// TwinCAT 3 PLC project TcpIp_SERVER_with_TLS_PSK
// Title: TLS Sample
// Company: Beckhoff Automation
// ProjectVersion: 1.0.0.0
// ProgramVersion: 3.1.0.5
// libraries:
//   Tc2_Standard, * (Beckhoff Automation GmbH)
//   Tc2_System, * (Beckhoff Automation GmbH)
//   Tc2_TcpIp, * (Beckhoff Automation GmbH)
//   Tc2_Utilities, * (Beckhoff Automation GmbH)
//   Tc3_Module, * (Beckhoff Automation GmbH)
// project tree:
//   Data types/ E_ConnectionSteps.TcDUT (not stored), E_ServerSteps.TcDUT
//   Global Variables/ Global_Variables.TcGVL
//   POUs/ FB_Server.TcPOU, FB_ServerApplication.TcPOU, FB_ServerConnection.TcPOU, MAIN.TcPOU
//   POUs/Helper POUs/ FB_FrameFifo.TcPOU (not stored), FB_LogFifo.TcPOU (not stored), FB_TlsConfig.TcPOU
//   / PlcTaskServer.TcTTO
// real-time tasks:
//   TASK PlcTaskServer: cycle T#10ms, priority 20, ADS port 350

CONFIGURATION TcpIp_SERVER_with_TLS_PSK
    RESOURCE PLC ON TwinCAT3
        TASK PlcTaskServer(INTERVAL := T#10ms, PRIORITY := 20);
        PROGRAM MAIN WITH PlcTaskServer : MAIN;
    END_RESOURCE
END_CONFIGURATION

// ---- Data types/E_ServerSteps.TcDUT
TYPE E_ServerSteps :
(
	eSERVER_STATE_IDLE,
	eSERVER_STATE_SOCKET_CREATE,
	eSERVER_STATE_LISTENER_OPEN_START,
	eSERVER_STATE_LISTENER_OPEN_WAIT,
	eSERVER_STATE_REMOTE_CLIENTS_COMM,
	eSERVER_STATE_REMOTE_CLIENTS_CLOSE,
	eSERVER_STATE_LISTENER_CLOSE_START,
	eSERVER_STATE_LISTENER_CLOSE_WAIT,
	eSERVER_STATE_ERROR
);
END_TYPE

// ---- Global Variables/Global_Variables.TcGVL
VAR_GLOBAL CONSTANT
	MAX_CLIENT_CONNECTIONS					: UDINT(1..20) := 5;
	PLCPRJ_BUFFER_SIZE						: UDINT := 1000;(* Max. internal fifo/receiver buffer size *)

(*	PLCPRJ_CLIENT_SEND_CYCLE_TIME			: TIME := T#1S; not used at server side *)
	PLCPRJ_RECEIVE_POLLING_TIME				: TIME := T#100MS;
	PLCPRJ_RECEIVE_TIMEOUT					: TIME := T#50S;

	(* Some project specific error codes *)
	PLCPRJ_ERROR_RECEIVE_TIMEOUT			: UDINT := 16#8101;(* Receive timeout *)
	PLCPRJ_ERROR_SENDFIFO_OVERFLOW			: UDINT := 16#8102;(* Send fifo overflow *)
	PLCPRJ_ERROR_RECFIFO_OVERFLOW			: UDINT := 16#8103;(* Receive fifo overflow *)
END_VAR

// ---- POUs/MAIN.TcPOU
PROGRAM MAIN
VAR
	sSrvNetID   : T_AmsNetID :='';(* TwinCAT TCP/IP server network address *)
	{warning 'Please configure your server IP-address and server port number below:'}
	sLocalHost  : T_IPv4Addr :='127.0.0.1';(*Own (server) IP address! *)
	nLocalPort  : UINT       :=200;(* Own (server) port number! *)
	
	bEnable     : BOOL       :=TRUE;(* TRUE => Enable server data exchange, FALSE => Disable *)
	bLog        : BOOL       :=TRUE;(* TRUE => Enable message/error log, FALSE => Disable *)
	
	bPSK        : BOOL       :=TRUE;(* TRUE => use PSK , FALSE => don't use PSK *)
	key         : ARRAY[0..14] OF BYTE:=[16#1B,16#D0,16#6F,16#D2,16#56,16#16,16#7D,16#C1,16#E8,16#C7,16#48,16#2A,16#8E,16#F5,16#FF];
	fbTls       : FB_TlsConfig;(* TLS/PSK configuration *)
	
	fbServer    : FB_Server:=(sLocalHost:=sLocalHost, nLocalPort:=nLocalPort, sPrefix:='SERVER::');
	fbCloseAll  : FB_SocketCloseAll;
	bInitialize : BOOL:=TRUE;
END_VAR

IF bInitialize THEN
	(* On PLC reset or program download close all created/opened sockets/connections *)
	fbCloseAll(sSrvNetID:=sSrvNetID, bExecute:=bInitialize);
	IF fbCloseAll.bBusy OR fbCloseAll.bError THEN
		RETURN;
	END_IF
	
	(* Configure TLS/PSK settings *)
	fbTls.Clear();
	IF bPSK THEN
		fbTls.AddPsk(key:=key, sIdentity:='MyIdentity');
	END_IF
	
	bInitialize:=FALSE;
END_IF

fbServer(fbTls:=fbTls, sSrvNetID:=sSrvNetID, bEnable:=bEnable, bLog:=bLog);

END_PROGRAM

// ---- POUs/Helper POUs/FB_TlsConfig.TcPOU
(* TLS/PSK configuration *)
{attribute 'no_explicit_call':='Direct call not allowed for type FB_TlsConfig'}
{attribute 'no_assign'}
FUNCTION_BLOCK FB_TlsConfig
VAR
	_pskKey       : ARRAY[0..TCPADS_TLS_MAX_PSK_KEY_SIZE] OF BYTE;
	_pskKeyLen    : UDINT:=0;
	_sIdentity    : STRING(TCPADS_TLS_PSK_IDENTITY_SIZE);
	_sCaPath      : STRING(TCPADS_TLS_CERTIFICATE_PATH_SIZE);
	_sCrlPath     : STRING(TCPADS_TLS_CERTIFICATE_PATH_SIZE);
	_sCertPath    : STRING(TCPADS_TLS_CERTIFICATE_PATH_SIZE);
	_sKeyPath     : STRING(TCPADS_TLS_CERTIFICATE_PATH_SIZE);
	_sKeyPwd      : STRING(TCPADS_TLS_KEY_PASSWORD_SIZE);
	_listenFlags  : ST_TlsListenFlags:=DEFAULT_TLSLISTENFLAGS;
	_connectFlags : ST_TlsConnectFlags:=DEFAULT_TLSCONNECTFLAGS;
END_VAR

(* Adds CA certificate path *)
METHOD FINAL AddCa
VAR_INPUT
	sCaPath : STRING(TCPADS_TLS_CERTIFICATE_PATH_SIZE);
END_VAR
_sCaPath:=sCaPath;
END_METHOD

(* Adds certificate path *)
METHOD FINAL AddCert
VAR_INPUT
	sCertPath: STRING(TCPADS_TLS_CERTIFICATE_PATH_SIZE);
	sKeyPath: STRING(TCPADS_TLS_CERTIFICATE_PATH_SIZE);
	sKeyPwd: STRING(TCPADS_TLS_KEY_PASSWORD_SIZE);
END_VAR
_sCertPath:=sCertPath;
_sKeyPath:=sKeyPath;
_sKeyPwd:=sKeyPwd;
END_METHOD

METHOD FINAL AddConnectFlags
VAR_INPUT
	flags : ST_TlsConnectFlags;
END_VAR
_connectFlags:=flags;
END_METHOD

(* Adds certificate revocation list path *)
METHOD FINAL AddCrl
VAR_INPUT
	sCrlPath : STRING(TCPADS_TLS_CERTIFICATE_PATH_SIZE);
END_VAR
_sCrlPath:=sCrlPath;
END_METHOD

METHOD FINAL AddListenFlags
VAR_INPUT
	flags : ST_TlsListenFlags;
END_VAR
_listenFlags:=flags;
END_METHOD

(* Adds PSK and PSK identity *)
METHOD FINAL AddPsk
VAR_IN_OUT
	key : ARRAY[*] OF BYTE;
END_VAR
VAR_INPUT
	sIdentity : STRING(TCPADS_TLS_PSK_IDENTITY_SIZE);
END_VAR
_pskKeyLen:=MIN(DINT_TO_UDINT(UPPER_BOUND(key, 1) - LOWER_BOUND(key, 1) + 1), TCPADS_TLS_MAX_PSK_KEY_SIZE, SIZEOF(_pskKey));
MEMCPY(ADR(_pskKey[0]), ADR(key[LOWER_BOUND(key, 1)]), _pskKeyLen);
_sIdentity:=sIdentity;
END_METHOD

METHOD FINAL Clear
_sIdentity:='';
_pskKeyLen:=0;
MEMSET(ADR(_pskKey[0]), 0, SIZEOF(_pskKey));
_sCaPath:='';
_sCertPath:='';
_sKeyPath:='';
_sKeyPwd:='';
_sCrlPath:='';
END_METHOD

PROPERTY FINAL connectFlags : ST_TlsConnectFlags
GET
connectFlags:=_connectFlags;
END_GET
END_PROPERTY

PROPERTY FINAL listenFlags : ST_TlsListenFlags
GET
listenFlags:=_listenFlags;
END_GET
END_PROPERTY

(* Pointer to first PSK key byte *)
PROPERTY FINAL pskKey : PVOID
GET
pskKey:=SEL(_pskKeyLen = 0, ADR(_pskKey[0]), 0);
END_GET
END_PROPERTY

(* Byte size of PSK key *)
PROPERTY FINAL pskKeyLen : UDINT(0..TCPADS_TLS_MAX_PSK_KEY_SIZE)
GET
pskKeyLen:=_pskKeyLen;
END_GET
END_PROPERTY

(* CA certificate path *)
PROPERTY FINAL sCaPath : STRING(TCPADS_TLS_CERTIFICATE_PATH_SIZE)
GET
sCaPath:=_sCaPath;
END_GET
END_PROPERTY

(* Certificate path *)
PROPERTY FINAL sCertPath : STRING(TCPADS_TLS_CERTIFICATE_PATH_SIZE)
GET
sCertPath:=_sCertPath;
END_GET
END_PROPERTY

(* Certificate revocation list path *)
PROPERTY FINAL sCrlPath : STRING(TCPADS_TLS_CERTIFICATE_PATH_SIZE)
GET
sCrlPath:=_sCrlPath;
END_GET
END_PROPERTY

(* PSK key identity *)
PROPERTY FINAL sIdentity : STRING(TCPADS_TLS_PSK_IDENTITY_SIZE)
GET
sIdentity:=_sIdentity;
END_GET
END_PROPERTY

(* Certificate key path *)
PROPERTY FINAL sKeyPath : STRING(TCPADS_TLS_CERTIFICATE_PATH_SIZE)
GET
sKeyPath:=_sKeyPath;
END_GET
END_PROPERTY

(* Certificate key password *)
PROPERTY FINAL sKeyPwd : STRING(TCPADS_TLS_KEY_PASSWORD_SIZE)
GET
sKeyPwd:=_sKeyPwd;
END_GET
END_PROPERTY

END_FUNCTION_BLOCK

// ---- POUs/FB_Server.TcPOU
FUNCTION_BLOCK FB_Server
VAR_IN_OUT
	fbTls          : FB_TlsConfig;(* TLS/PSK configuration *)
END_VAR
VAR_INPUT
	sSrvNetID      : T_AmsNetID :='';(* TwinCAT TCP/IP server network address *)
	sLocalHost     : T_IPv4Addr :='127.0.0.1';(* Own IP address! *)
	nLocalPort     : UDINT      :=0;(* Server port number *)
	bEnable        : BOOL       :=FALSE;(* TRUE => enable server data exchange, FALSE => disable *)
	tReconnect     : TIME       :=T#3S;(* Reopen new listener socket after this time *)
	bLog           : BOOL       :=FALSE;(* TRUE => Enable log message output, FALSE => Disable *)
	sPrefix        : STRING     :='SERVER::';(* Log message description string (allows the identification of log message source) *)
END_VAR
VAR_OUTPUT
	bListening     : BOOL       :=FALSE;(* Listener socket state *)
	nAccepted      : UDINT      :=0;(* Max. number of accepted client connections *)
END_VAR
VAR
	aApplications  : ARRAY[1..MAX_CLIENT_CONNECTIONS] OF FB_ServerApplication;(* Server application control function blocks *)
	aConnections   : ARRAY[1..MAX_CLIENT_CONNECTIONS] OF FB_ServerConnection :=[
														(sPrefix := 'SERVER1::'),
														(sPrefix := 'SERVER2::'),
														(sPrefix := 'SERVER3::'),
														(sPrefix := 'SERVER4::'),
														(sPrefix := 'SERVER5::')];(* Server connection/data exchange control function blocks *)
	aTx            : ARRAY[1..MAX_CLIENT_CONNECTIONS] OF FB_FrameFifo;(* TX fifo *)
	aRx            : ARRAY[1..MAX_CLIENT_CONNECTIONS] OF FB_FrameFifo;(* RX fifo *)
	aLog           : ARRAY[1..MAX_CLIENT_CONNECTIONS] OF FB_LogFifo;(* Listener log message fifo *)

	fbCreate       : FB_TlsSocketCreate:=(bListener:=TRUE);(* Creates listener socket *)
	fbListen       : FB_TlsSocketListen;(* Opens listener socket *)
	fbSetPsk       : FB_TlsSocketSetPsk;(* Configures PSK (pre-shared key) *)
	fbClose        : FB_SocketClose;(* Closes socket *)
	fbLog          : FB_LogFifo;
	fbListenTimer  : TON;
	bReset         : BOOL :=FALSE;
	eStep          : E_ServerSteps;
	i              : UDINT;
END_VAR

CASE eStep OF
	eSERVER_STATE_IDLE:
		IF bEnable XOR bListening THEN
			IF bEnable THEN
				fbListenTimer( IN := TRUE );
				IF fbListenTimer.Q THEN
					fbListenTimer( IN := FALSE, PT := tReconnect );

					fbLog.Clear( sPrefix := sPrefix, bLog := bLog );(* Clear listener log fifo *)
					bReset := FALSE;

					fbCreate(bExecute:=FALSE);
					fbCreate(sSrvNetID:=sSrvNetID, bExecute:=TRUE);
					eStep := eSERVER_STATE_SOCKET_CREATE;
				END_IF
			ELSE
				eStep := eSERVER_STATE_REMOTE_CLIENTS_CLOSE;
			END_IF
		ELSIF bListening THEN
			eStep := eSERVER_STATE_REMOTE_CLIENTS_COMM;
		ELSE
			fbListenTimer( IN := FALSE, PT := T#0S );
			bReset := FALSE;
		END_IF
		
	eSERVER_STATE_SOCKET_CREATE:
		fbCreate(bExecute:=FALSE);
		IF NOT fbCreate.bBusy THEN
			IF NOT fbCreate.bError THEN
				fbSetPsk(bExecute:=FALSE);
				IF (fbTls.pskKeyLen <> 0) AND (fbTls.pskKey <> 0) AND (fbTls.sIdentity <> '') THEN
					fbSetPsk(sSrvNetID:=sSrvNetID, hSocket:=fbCreate.hSocket, sIdentity:=fbTls.sIdentity, pskKey:=fbTls.pskKey, pskKeyLen:=fbTls.pskKeyLen, bExecute:=TRUE);
				END_IF
				eStep := eSERVER_STATE_LISTENER_OPEN_START;
			ELSE
				fbLog.Error( sMessage := 'FB_TlsSocketCreate()', nErrId := fbCreate.nErrId);
				eStep := eSERVER_STATE_ERROR;
			END_IF
		END_IF

	eSERVER_STATE_LISTENER_OPEN_START:
		fbSetPsk(bExecute:=FALSE);
		IF NOT fbSetPsk.bBusy THEN
			IF NOT fbSetPsk.bError THEN
				fbListen(bExecute:=FALSE, hListener:=fbCreate.hSocket);
				fbListen(sSrvNetID:=sSrvNetID, bExecute:=TRUE, hListener:=fbCreate.hSocket, sLocalHost:=sLocalHost, nLocalPort:=nLocalPort);
				eStep := eSERVER_STATE_LISTENER_OPEN_WAIT;
			ELSE
				fbLog.Error( sMessage := 'FB_TlsSocketSetPsk()', nErrId := fbSetPsk.nErrId);
				eStep := eSERVER_STATE_ERROR;
			END_IF
		END_IF

	eSERVER_STATE_LISTENER_OPEN_WAIT:
		fbListen(bExecute:=FALSE, hListener:=fbCreate.hSocket);
		IF NOT fbListen.bBusy THEN
			IF NOT fbListen.bError THEN
				bListening := TRUE;
				fbLog.Message( sMessage := 'Listener socket opened!', hSocket := fbCreate.hSocket);
				eStep := eSERVER_STATE_IDLE;
			ELSE
				fbLog.Error( sMessage := 'FB_TlsSocketListen()', nErrId := fbListen.nErrId );
				eStep := eSERVER_STATE_ERROR;
			END_IF
		END_IF

	eSERVER_STATE_REMOTE_CLIENTS_COMM:
		eStep := eSERVER_STATE_IDLE;
		nAccepted := 0;

		FOR i:= 1 TO MAX_CLIENT_CONNECTIONS DO
			aConnections[i]( fbTx := aTx[i], fbRx := aRx[i], fbLog := aLog[i],
							hListener := fbCreate.hSocket, bReset := bReset,
							sSrvNetID := sSrvNetID, bEnable := bEnable,	bLog := bLog );
			IF bReset THEN
				bReset := FALSE;
				eStep := eSERVER_STATE_REMOTE_CLIENTS_CLOSE;
				EXIT;
			END_IF
			
			IF aConnections[i].bAccepted THEN
				aApplications[i]( fbTx := aTx[i], fbRx := aRx[i], fbLog := aLog[i] );
				nAccepted := nAccepted + 1;(* Count the number of connected remote clients *)
			END_IF

		END_FOR

	eSERVER_STATE_REMOTE_CLIENTS_CLOSE:
		nAccepted := 0;
		FOR i:= 1 TO MAX_CLIENT_CONNECTIONS DO
			(* Close all remote client (accepted) sockets *)
			aConnections[i]( fbTx := aTx[i], fbRx := aRx[i], fbLog := aLog[i],
							hListener := fbCreate.hSocket, bReset := bReset,
							sSrvNetID := sSrvNetID, bEnable := FALSE, bLog := bLog );
			IF aConnections[i].bAccepted THEN
				nAccepted := nAccepted + 1;(* Count the number of connected remote clients *)
			END_IF
		END_FOR
		
		(* Check if all remote client sockets are closed *)
		IF nAccepted = 0 THEN
			eStep := eSERVER_STATE_LISTENER_CLOSE_START; (* Close listener socket too *)
		END_IF

	eSERVER_STATE_LISTENER_CLOSE_START:
		fbLog.Message( sMessage := 'Closing listener socket!', hSocket := fbCreate.hSocket);
		fbClose(bExecute:=FALSE);
		fbClose(sSrvNetID:=sSrvNetID, hSocket:=fbCreate.hSocket, bExecute:=TRUE);
		eStep := eSERVER_STATE_LISTENER_CLOSE_WAIT;

	eSERVER_STATE_LISTENER_CLOSE_WAIT:
		fbClose( bExecute := FALSE );
		IF NOT fbClose.bBusy THEN
			bListening := FALSE;
			nAccepted := 0;
			IF NOT fbClose.bError THEN
				eStep := eSERVER_STATE_IDLE;
			ELSE
				fbLog.Error( sMessage := 'FB_SocketClose(listener)', nErrId := fbListen.nErrID );
				eStep := eSERVER_STATE_ERROR;
			END_IF
		END_IF

	eSERVER_STATE_ERROR:
		IF bListening THEN
			eStep := eSERVER_STATE_REMOTE_CLIENTS_CLOSE;
		ELSE
			eStep := eSERVER_STATE_IDLE;
		END_IF

END_CASE

END_FUNCTION_BLOCK

// ---- POUs/FB_ServerApplication.TcPOU
(*------------- Simple TCP/IP server application. Adapt this code to match your needs. -----*)
FUNCTION_BLOCK FB_ServerApplication
VAR_IN_OUT
	fbTx        : FB_FrameFifo;(* TX fifo *)
	fbRx        : FB_FrameFifo;(* RX fifo *)
	fbLog       : FB_LogFifo;(* Log message fifo *)
END_VAR
VAR
	sToClient   : T_MaxString:='';
	sFromClient : T_MaxString:='';
	sLogMessage : T_MaxString:='';
	nCounter    : UDINT;
END_VAR

(*------------------------------- Get received message strings ---------------------------------*)
REPEAT
	fbRx.RemoveHead( );(* Fetch string from rx fifo *)
	IF fbRx.bOk THEN(* Success *)

		(* TODO: Implement receive message handler *)
		(* Example: Send message strings back to the client *)

	
		nCounter := nCounter + 1;
	
		sFromClient := fbRx.sGet;
		sToClient := sFromClient;
	
		fbTx.AddTail( sPut := sToClient );(* Put string to the tx fifo *)
		IF NOT fbTx.bOk THEN(* TX fifo overflow => log error *)
			fbLog.Error( sMessage := 'FB_FrameFifo(sender)', nErrID := PLCPRJ_ERROR_SENDFIFO_OVERFLOW ); 
		END_IF
		
	END_IF
UNTIL NOT fbRx.bOk
END_REPEAT

(*------------------------------- Get log/error messages from log fifo ---------------------------*)
REPEAT
	fbLog.Remove( );
	IF fbLog.bOk THEN(* Success *)
		
		(* TODO: Implement log message handler *)
		sLogMessage := fbLog.sGet;
		
	END_IF
UNTIL NOT fbLog.bOk
END_REPEAT

END_FUNCTION_BLOCK

// ---- POUs/FB_ServerConnection.TcPOU
FUNCTION_BLOCK FB_ServerConnection
VAR_IN_OUT
	fbTx            : FB_FrameFifo;(* TX fifo *)
	fbRx            : FB_FrameFifo;(* RX fifo *)
	fbLog           : FB_LogFifo;(* Log message fifo *)
	hListener       : T_HSOCKET;(* Listener socket handle *)
	bReset          : BOOL;
END_VAR
VAR_INPUT
	sSrvNetID       : T_AmsNetID :='';(* TwinCAT TCP/IP server network address *)
	bEnable         : BOOL       :=FALSE;(* TRUE => connect and exchange data, FALSE => disconnect *)
	tReconnect      : TIME       :=T#1S;(* Accept new connection (reconnect) after this time *)
	bLog            : BOOL       :=FALSE;(* TRUE => Enable log message output, FALSE => Disable *)
	sPrefix         : STRING     :='SERVERx::';(* Log message description string (allows the identification of log message source) *)
END_VAR
VAR_OUTPUT
	bAccepted       : BOOL       :=FALSE;(* Accepted connection status *)
END_VAR
VAR
	fbAccept        : FB_SocketAccept;(* Accepts new server connection *)
	fbClose         : FB_SocketClose;(* Closes accepted connection *)
	fbReceive       : FB_SocketReceive;(* Receives data *)
	fbSend          : FB_SocketSend;(* Sends data *)
	eStep           : E_ConnectionSteps;
	bSndBusy        : BOOL;(* Tx state *)
	bRcvBusy        : BOOL;(* Rx state *)
	bDisconnect     : BOOL;(* Disconnect flag, if set the socket will be closed *)

	fbAcceptTimer   : TON;(* Accept poll timer *)
	fbPollTimer     : TON;(* Receive poll timer *)
	fbRequestTimer  : TON;(* Request timeout timer *)
	
	rxBuffer        : ARRAY[0..PLCPRJ_BUFFER_SIZE] OF BYTE;
	sTxFrame        : T_MaxString;
	sRxFrame        : T_MaxString;
	cbReceived      : UDINT;
	nLenOfString    : UDINT;(* String length inclusive the null delimiter *)
	bEndOfString    : BOOL:=FALSE;
END_VAR

CASE eStep OF
	eCONNECTION_STATE_IDLE:
		IF bEnable XOR bAccepted THEN
			IF bEnable THEN
				fbAcceptTimer( IN := TRUE );
				IF fbAcceptTimer.Q THEN
					
					fbTx.Clear( sPrefix := CONCAT( sPrefix, 'FB_FrameFifo(sender)::' ), bLog := bLog );(* Clear send fifo *)
					fbRx.Clear( sPrefix := CONCAT( sPrefix, 'FB_FrameFifo(receiver)::' ), bLog := bLog );(* Clear receiver fifo *)
					fbLog.Clear( sPrefix := sPrefix, bLog := bLog );(* Clear log fifo *)
					bSndBusy := FALSE;
					bRcvBusy := FALSE;
					bDisconnect := FALSE;
					cbReceived := 0;
					
					fbPollTimer( IN := FALSE, PT := T#0S );
					fbRequestTimer( IN := FALSE, PT := PLCPRJ_RECEIVE_TIMEOUT );
					fbAcceptTimer( IN := FALSE, PT := tReconnect );
					
					
					eStep := eCONNECTION_STATE_CONNECT_START;
				END_IF
			ELSE
				eStep := eCONNECTION_STATE_CLOSE_START;
			END_IF
		ELSIF bAccepted THEN
			eStep := eCONNECTION_STATE_DATAEXCHANGE;
		ELSE
			fbAcceptTimer( IN := FALSE, PT := T#0S );
		END_IF

	eCONNECTION_STATE_CONNECT_START:
		fbAccept( bExecute := FALSE );
		fbAccept( sSrvNetID := sSrvNetID,
					hListener := hListener,
					bExecute:= TRUE );
		eStep := eCONNECTION_STATE_CONNECT_WAIT;

	eCONNECTION_STATE_CONNECT_WAIT:
		fbAccept( bExecute := FALSE );
		IF NOT fbAccept.bBusy THEN
			IF NOT fbAccept.bError THEN
				IF fbAccept.bAccepted THEN
					bAccepted := TRUE;
					fbLog.Message( sMessage := 'Connection accepted!', hSocket := fbAccept.hSocket );
				END_IF
				eStep := eCONNECTION_STATE_IDLE;
			ELSE
				fbLog.Error( sMessage := 'FB_SocketAccept()', nErrId := fbAccept.nErrId );
				eStep := eCONNECTION_STATE_ERROR;
			END_IF
		END_IF

	eCONNECTION_STATE_DATAEXCHANGE:(* Data exchange state *)
		bDisconnect := NOT bEnable OR bDisconnect;(* User/internal disconnect requested? *)
		IF bDisconnect AND NOT bSndBusy AND NOT bRcvBusy THEN
			bDisconnect := FALSE;
			eStep := eCONNECTION_STATE_CLOSE_START;(* Disconnect *)
		ELSE
	
			(* Send tx data *)
			IF NOT bDisconnect AND NOT bSndBusy THEN
				fbTx.RemoveHead( sGet => sTxFrame );(* Remove oldest string entry s*)
				IF fbTx.bOk THEN(* Success *)
					fbSend( bExecute := FALSE );
					fbSend(	sSrvNetID := sSrvNetID, 
							hSocket	:= fbAccept.hSocket,
							pSrc	:= ADR( sTxFrame ),
							cbLen	:= INT_TO_UDINT(LEN( sTxFrame )) + 1,(* String length inclusive the zero delimiter *)
							bExecute:= TRUE );
					bSndBusy := TRUE;
				END_IF
			ELSE
				fbSend( bExecute := FALSE );
				IF NOT fbSend.bBusy THEN
					bSndBusy := FALSE;
					IF fbSend.bError THEN
						fbLog.Error( sMessage := 'FB_SocketSend()', nErrId := fbSend.nErrId );
						bDisconnect := TRUE;(* Set flag *)
					END_IF
				END_IF
			END_IF
		
		
			(* Get rx data *)
			IF NOT bDisconnect AND NOT bRcvBusy THEN
				fbPollTimer( IN := TRUE );
				IF fbPollTimer.Q THEN
					fbPollTimer( IN := FALSE, PT := PLCPRJ_RECEIVE_POLLING_TIME );
					fbReceive( bExecute := FALSE );
					fbReceive( 	sSrvNetID := sSrvNetID,
								hSocket	:= fbAccept.hSocket,
								pDest	:= ADR( rxBuffer ) + cbReceived,
								cbLen	:= SIZEOF( rxBuffer ) - cbReceived,
								bExecute:= TRUE );
					bRcvBusy := TRUE;
				END_IF
			ELSE
				fbReceive( bExecute := FALSE );
				IF NOT fbReceive.bBusy THEN
					bRcvBusy := FALSE;
					IF NOT fbReceive.bError THEN
						IF (fbReceive.nRecBytes > 0) THEN(* Bytes received *)
							
							fbPollTimer( IN := FALSE, PT := T#0S ); (* Bytes received => increase the read (polling) speed *)
							fbRequestTimer( IN := FALSE );(* Bytes received => disable timeout check *)
							cbReceived 	:= cbReceived + fbReceive.nRecBytes;(* Calculate the number of received data bytes *)
		
							REPEAT
								
								(* Search for string end delimiter *)
								nLenOfString := 0;(* Reset string length *)
								bEndOfString := FALSE;
								REPEAT 
									IF rxBuffer[nLenOfString] = 0 THEN(* String end delimiter found *)
										bEndOfString := TRUE;
									END_IF
									nLenOfString := nLenOfString + 1;
								UNTIL bEndOfString OR (nLenOfString >= cbReceived)
								END_REPEAT
								
								IF bEndOfString THEN
									MEMSET( ADR( sRxFrame ), 0, SIZEOF( sRxFrame ) );
									MEMCPY(  ADR( sRxFrame ), ADR( rxBuffer ), MIN( SIZEOF(sRxFrame), nLenOfString ) );(* Copy the received string to the output variable (inclusive the end delimiter) *)
									MEMMOVE( ADR( rxBuffer ), ADR( rxBuffer[nLenOfString] ), cbReceived - nLenOfString  );(* Move the reamaining data bytes *)
									cbReceived := cbReceived - nLenOfString;(* Recalculate the reamaining data byte length *)
			
									fbRx.AddTail( sPut := sRxFrame );(* Put received message to the rx fifo *)
									IF NOT fbRx.bOk THEN
										fbLog.Error( sMessage := 'FB_FrameFifo(receiver)', nErrID := PLCPRJ_ERROR_RECFIFO_OVERFLOW );
										bDisconnect := TRUE;(* Set flag *)
										RETURN;
									END_IF
								END_IF

							UNTIL NOT bEndOfString OR (cbReceived = 0)
							END_REPEAT
		
						ELSE(* No bytes received *)
							fbRequestTimer( IN := TRUE, PT := PLCPRJ_RECEIVE_TIMEOUT );(* No bytes received => enable timeout check *)
							IF fbRequestTimer.Q THEN (* Timeout error*)
								fbRequestTimer( IN := FALSE );
								fbLog.Error( sMessage := 'FB_SocketReceive()', nErrID := PLCPRJ_ERROR_RECEIVE_TIMEOUT );
								bDisconnect := TRUE;(* Set flag *)
							END_IF
						END_IF
						
					ELSE(* Receive error *)
						fbLog.Error( sMessage := 'FB_SocketReceive()', nErrId := fbReceive.nErrId );
						bDisconnect := TRUE;(* Set flag *)
					END_IF
				END_IF(* IF NOT fbReceive.bBusy THEN *)
				
			END_IF(* IF NOT bDisconnect AND NOT bRcvBusy THEN *)
		
		END_IF(* IF bDisconnect AND NOT bSndBusy AND NOT bRcvBusy THEN *)
	
	

	eCONNECTION_STATE_CLOSE_START:
		fbLog.Message( sMessage := 'Closing connection!', hSocket := fbAccept.hSocket );
		fbClose( bExecute := FALSE );
		fbClose( sSrvNetID := sSrvNetID, hSocket:= fbAccept.hSocket, bExecute:= TRUE );
		eStep := eCONNECTION_STATE_CLOSE_WAIT;

	eCONNECTION_STATE_CLOSE_WAIT:
		fbClose( bExecute := FALSE );
		IF NOT fbClose.bBusy THEN
			bAccepted := FALSE;
			IF NOT fbClose.bError THEN
				eStep := eCONNECTION_STATE_IDLE;
			ELSE
				fbLog.Error( sMessage := 'FB_SocketClose(accepted)', nErrId := fbClose.nErrId );
				eStep := eCONNECTION_STATE_ERROR;
			END_IF
		END_IF

	eCONNECTION_STATE_ERROR:
		IF bAccepted THEN
			eStep := eCONNECTION_STATE_CLOSE_START;
		ELSE
			eStep := eCONNECTION_STATE_IDLE;
		END_IF

END_CASE

END_FUNCTION_BLOCK
